// TIA Portal project "Funcoes" (V18)

(* hardware
DEVICE "S7-1200 station_1"  S7-1200 Station
   slot 0: "Rack_0"  S7-1200 Rack  Rack  V1.0
   slot 1: "PLC_1"  CPU 1214C AC/DC/Rly  6ES7 214-1BG40-0XB0  V4.5
   slot 2: "DI 16/DQ 16x24VDC_1"  6ES7 223-1BL32-0XB0  V2.0
   slot 3: "AI 8x13BIT_1"  6ES7 231-4HF32-0XB0  V2.1
*)

// ===== PLC "PLC_1"  CPU 1214C AC/DC/Rly =====

VAR_GLOBAL   // PLC tag table "Default tag table"
   "VC" AT %Q0.0 : Bool;
   "VT" AT %Q0.1 : Bool;
   "VD1" AT %Q0.2 : Bool;
   "VD2" AT %Q0.3 : Bool;
   "C1" AT %Q0.4 : Bool;
   "C2" AT %Q0.5 : Bool;
   "C3" AT %Q0.6 : Bool;
   "LED1" AT %Q0.7 : Bool;
   "LED2" AT %Q1.0 : Bool;
   "LE" AT %Q1.1 : Bool;
   "H" AT %Q8.0 : Bool;
   "BL" AT %I0.0 : Bool;
   "BD" AT %I0.1 : Bool;
   "BE" AT %I0.2 : Bool;
   "CS1" AT %I0.3 : Bool;
   "CS2" AT %I0.4 : Bool;
   "P" AT %IW112 : Int;
   "PS" AT %IW114 : Int;
   "PA" AT %IW116 : Int;
   "T" AT %IW118 : Int;
END_VAR

VAR_GLOBAL CONSTANT   // PLC tag table "Default tag table"
   "Lmin" : Real := 1.0;
   "L1" : Real := 1.5;
   "L2" : Real := 2.0;
   "Tlim" : Real := 0.6;
   "Ta" : Real := 2.0;
   "beta" : Real := 0.02;
   "Padm" : Real := 3.5;
   "Pmin" : Real := 0.1;
   "Peq" : Real := 3.0;
   "gamma" : Real := 0.01;
   "Plim" : Real := 0.1;
END_VAR

DATA_BLOCK "Data_block_1"   // DB1
{ S7_Optimized_Access := 'TRUE' }
VERSION : 0.1
   VAR
      n : Int := 0;
      "Valvulas ON" : Bool := false;
      "Valvulas ON - M3" : Bool := false;
      "Sequencia 1" : Array[0..2] of Int;
      "Sequencia 2" : Array[0..2] of Int;
      "Sequencia 3" : Array[0..2] of Int;
   END_VAR
   VAR RETAIN
      Sequencia : Array[0..2] of Int;
   END_VAR
   VAR
      "Tomada de decisao" : Bool := false;
      "Valores de pressao" : Array[0..9] of Real;
      index : Int := 0;
      "index max" : Int := 10;
      length : Int := 10;
      "Valores de pressao - M3" : Array[0..999] of Real;
      "index - M3" : Int := 0;
      "index max - M3" : Int := 1000;
      "length - M3" : Int := 0;
      "Atingir pressao eq" : Bool := false;
      "Plim atingida" : Bool := false;
      M2 : Bool := false;
      "Estado anterior" : Bool := false;
   END_VAR
BEGIN
   "Sequencia 1"[0] := 1;
   "Sequencia 1"[1] := 2;
   "Sequencia 1"[2] := 3;
   "Sequencia 2"[0] := 3;
   "Sequencia 2"[1] := 1;
   "Sequencia 2"[2] := 2;
   "Sequencia 3"[0] := 2;
   "Sequencia 3"[1] := 3;
   "Sequencia 3"[2] := 1;
   Sequencia[0] := 1;
   Sequencia[1] := 2;
   Sequencia[2] := 3;
   "Valores de pressao"[0] := 0.0;
   "Valores de pressao"[1] := 0.0;
   "Valores de pressao"[2] := 0.0;
   "Valores de pressao"[3] := 0.0;
   "Valores de pressao"[4] := 0.0;
   "Valores de pressao"[5] := 0.0;
   "Valores de pressao"[6] := 0.0;
   "Valores de pressao"[7] := 0.0;
   "Valores de pressao"[8] := 0.0;
   "Valores de pressao"[9] := 0.0;
END_DATA_BLOCK

// folder: System blocks/Program resources

DATA_BLOCK "Timer de amostragem"   // DB2
{ S7_Optimized_Access := 'TRUE' }
AUTHOR : Simatic
FAMILY : IEC
NAME : IEC_TMR
VERSION : 1.0
// stored: InstanceOfName IEC_TIMER
"IEC_TIMER"
BEGIN
   PT := T#1S;
END_DATA_BLOCK

DATA_BLOCK "Timer abastecimento"   // DB3
{ S7_Optimized_Access := 'TRUE' }
AUTHOR : Simatic
FAMILY : IEC
NAME : IEC_TMR
VERSION : 1.0
// stored: InstanceOfName IEC_TIMER
"IEC_TIMER"
BEGIN
   PT := T#1S;
END_DATA_BLOCK

// folder: (top level)

FUNCTION "Aciona valvulas - M1 e M2" : Void   // FC1, LAD
{ S7_Optimized_Access := 'TRUE' }
VERSION : 0.1
BEGIN

REGION Network 1: Acionando válvulas dos modos 1 e 2
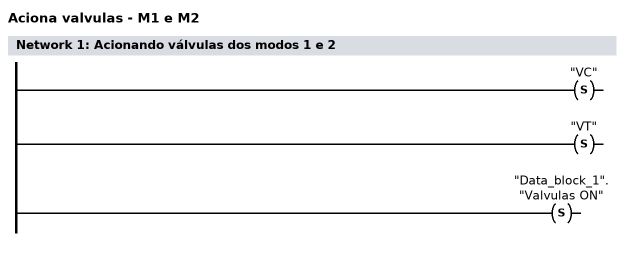
   RUNG wire#powerrail
      S_Coil( "VC" )
   END_RUNG
   RUNG wire#powerrail
      S_Coil( "VT" )
   END_RUNG
   RUNG wire#powerrail
      S_Coil( "Data_block_1"."Valvulas ON" )
   END_RUNG
   // the same network as SCL:
   "VC" := TRUE;
   "VT" := TRUE;
   "Data_block_1"."Valvulas ON" := TRUE;
END_REGION
END_FUNCTION

FUNCTION "Desliga valvulas - M1 e M2" : Void   // FC2, LAD
{ S7_Optimized_Access := 'TRUE' }
VERSION : 0.1
BEGIN

REGION Network 1: Válvula on/off da entrada do sistema de compressores
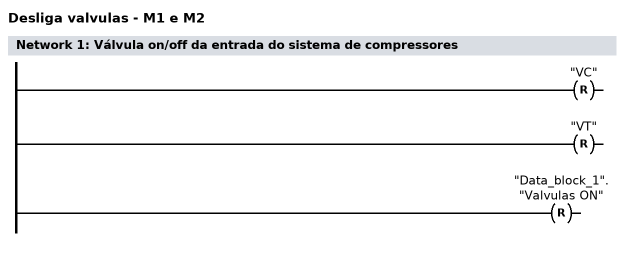
   RUNG wire#powerrail
      R_Coil( "VC" )
   END_RUNG
   RUNG wire#powerrail
      R_Coil( "VT" )
   END_RUNG
   RUNG wire#powerrail
      R_Coil( "Data_block_1"."Valvulas ON" )
   END_RUNG
   // the same network as SCL:
   "VC" := FALSE;
   "VT" := FALSE;
   "Data_block_1"."Valvulas ON" := FALSE;
END_REGION
END_FUNCTION

FUNCTION "Verifica valvulas 1" : Void   // FC3, LAD
{ S7_Optimized_Access := 'TRUE' }
VERSION : 0.1
BEGIN

REGION Network 1
   // Se válvulas OFF
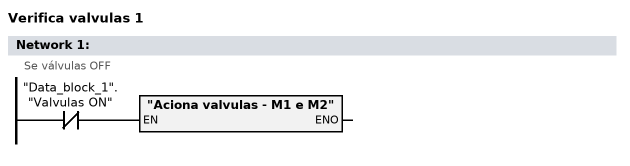
   RUNG wire#powerrail
      I_Contact( "Data_block_1"."Valvulas ON" )
      "Aciona valvulas - M1 e M2"()
   END_RUNG
   // the same network as SCL:
   IF NOT "Data_block_1"."Valvulas ON" THEN "Aciona valvulas - M1 e M2"(); END_IF;
END_REGION
END_FUNCTION

FUNCTION "Verifica valvulas 2" : Void   // FC4, LAD
{ S7_Optimized_Access := 'TRUE' }
VERSION : 0.1
BEGIN

REGION Network 1
   // Se válvulas ON
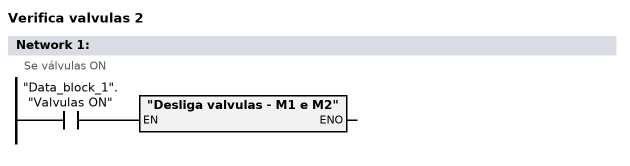
   RUNG wire#powerrail
      Contact( "Data_block_1"."Valvulas ON" )
      "Desliga valvulas - M1 e M2"()
   END_RUNG
   // the same network as SCL:
   IF "Data_block_1"."Valvulas ON" THEN "Desliga valvulas - M1 e M2"(); END_IF;
END_REGION
END_FUNCTION

FUNCTION "Obtem pressao" : Void   // FC5, LAD
{ S7_Optimized_Access := 'TRUE' }
VERSION : 0.1
   VAR_OUTPUT
      Pressao : Real;   // Pressão obtida
   END_VAR
   VAR_TEMP
      "Pressao normalizada" : Real;   // Pressão normalizada
   END_VAR
BEGIN

REGION Network 1
   // Normalização do valor de pressão lido do transmissor
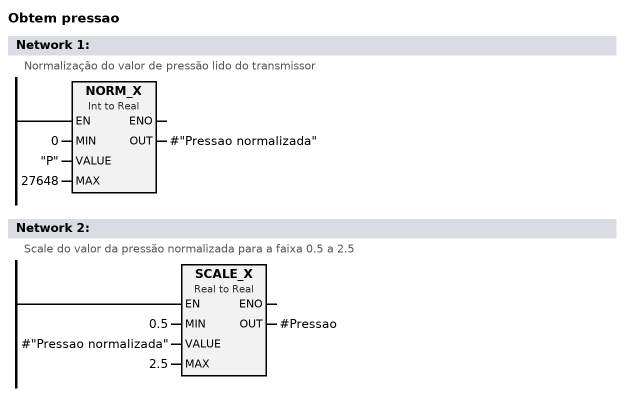
   RUNG wire#powerrail
      { S7_Templates := "[SrcType := Int, DestType := Real]" } Normalize(min := 0, value := "P", max := 27648, out => #"Pressao normalizada")
   END_RUNG
   // the same network as SCL:
   #"Pressao normalizada" := NORM_X(MIN := 0, VALUE := "P", MAX := 27648);
END_REGION

REGION Network 2
   // Scale do valor da pressão normalizada para a faixa 0.5 a 2.5
   RUNG wire#powerrail
      { S7_Templates := "[SrcType := Real, DestType := Real]" } Scale(min := 0.5, value := #"Pressao normalizada", max := 2.5, out => #Pressao)
   END_RUNG
   // the same network as SCL:
   #Pressao := SCALE_X(MIN := 0.5, VALUE := #"Pressao normalizada", MAX := 2.5);
END_REGION
END_FUNCTION

FUNCTION "Pressao crescente" : Void   // FC6, LAD
{ S7_Optimized_Access := 'TRUE' }
VERSION : 0.1
   VAR_INPUT
      P : Real;   // Pressão no interior do tanque separador
   END_VAR
   VAR_TEMP   // added for the SCL form of the ladder/FBD networks
      _w1 : Bool;
      _w2 : Bool;
   END_VAR
BEGIN

REGION Network 1
   // Se pressão entre Lmin e L1
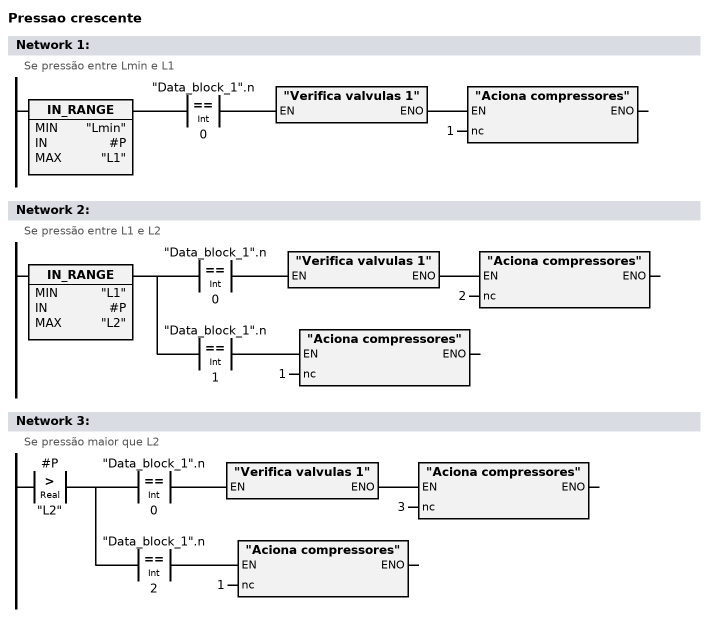
   RUNG wire#powerrail
      { S7_Templates := "SrcType := Real" } InRange(min := "Lmin", in := #P, max := "L1")
      { S7_Templates := "SrcType := Int" } EQ_Contact(in1 := "Data_block_1".n, in2 := 0)
      "Verifica valvulas 1"()
      "Aciona compressores"(nc := 1)
   END_RUNG
   // the same network as SCL:
   "Verifica valvulas 1"(EN := ("Lmin" <= #P) AND (#P <= "L1") AND ("Data_block_1".n = 0), ENO => #_w1);
   IF #_w1 THEN "Aciona compressores"(nc := 1); END_IF;
END_REGION

REGION Network 2
   // Se pressão entre L1 e L2
   RUNG wire#powerrail
      { S7_Templates := "SrcType := Real" } InRange(min := "L1", in := #P, max := "L2")
      wire#w1
      { S7_Templates := "SrcType := Int" } EQ_Contact(in1 := "Data_block_1".n, in2 := 0)
      "Verifica valvulas 1"()
      "Aciona compressores"(nc := 2)
   END_RUNG
   RUNG wire#w1
      { S7_Templates := "SrcType := Int" } EQ_Contact(in1 := "Data_block_1".n, in2 := 1)
      "Aciona compressores"(nc := 1)
   END_RUNG
   // the same network as SCL:
   #_w1 := ("L1" <= #P) AND (#P <= "L2");
   "Verifica valvulas 1"(EN := #_w1 AND ("Data_block_1".n = 0), ENO => #_w2);
   IF #_w2 THEN "Aciona compressores"(nc := 2); END_IF;
   IF #_w1 AND ("Data_block_1".n = 1) THEN "Aciona compressores"(nc := 1); END_IF;
END_REGION

REGION Network 3
   // Se pressão maior que L2
   RUNG wire#powerrail
      { S7_Templates := "SrcType := Real" } GT_Contact(in1 := #P, in2 := "L2")
      wire#w1
      { S7_Templates := "SrcType := Int" } EQ_Contact(in1 := "Data_block_1".n, in2 := 0)
      "Verifica valvulas 1"()
      "Aciona compressores"(nc := 3)
   END_RUNG
   RUNG wire#w1
      { S7_Templates := "SrcType := Int" } EQ_Contact(in1 := "Data_block_1".n, in2 := 2)
      "Aciona compressores"(nc := 1)
   END_RUNG
   // the same network as SCL:
   #_w1 := #P > "L2";
   "Verifica valvulas 1"(EN := #_w1 AND ("Data_block_1".n = 0), ENO => #_w2);
   IF #_w2 THEN "Aciona compressores"(nc := 3); END_IF;
   IF #_w1 AND ("Data_block_1".n = 2) THEN "Aciona compressores"(nc := 1); END_IF;
END_REGION
END_FUNCTION

FUNCTION "Pressao decrescente" : Void   // FC7, LAD
{ S7_Optimized_Access := 'TRUE' }
VERSION : 0.1
   VAR_INPUT
      P : Real;   // Pressão no interior do tanque separador
   END_VAR
   VAR_TEMP   // added for the SCL form of the ladder/FBD networks
      _w1 : Bool;
   END_VAR
BEGIN

REGION Network 1
   // Se pressão entre L1 e L2
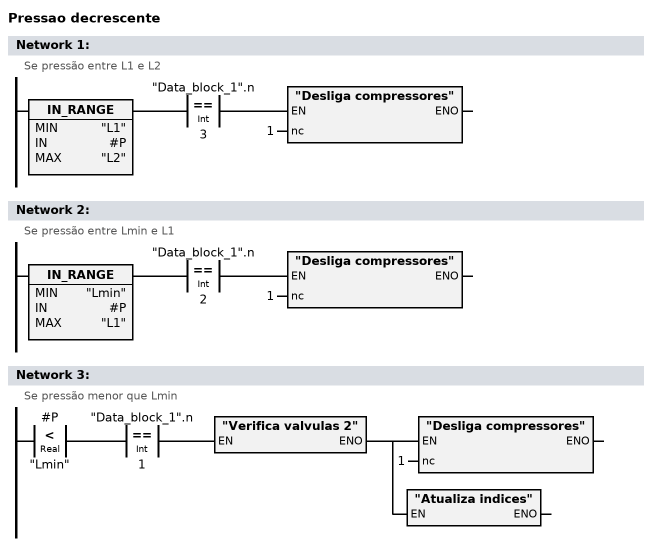
   RUNG wire#powerrail
      { S7_Templates := "SrcType := Real" } InRange(min := "L1", in := #P, max := "L2")
      { S7_Templates := "SrcType := Int" } EQ_Contact(in1 := "Data_block_1".n, in2 := 3)
      "Desliga compressores"(nc := 1)
   END_RUNG
   // the same network as SCL:
   IF ("L1" <= #P) AND (#P <= "L2") AND ("Data_block_1".n = 3) THEN "Desliga compressores"(nc := 1); END_IF;
END_REGION

REGION Network 2
   // Se pressão entre Lmin e L1
   RUNG wire#powerrail
      { S7_Templates := "SrcType := Real" } InRange(min := "Lmin", in := #P, max := "L1")
      { S7_Templates := "SrcType := Int" } EQ_Contact(in1 := "Data_block_1".n, in2 := 2)
      "Desliga compressores"(nc := 1)
   END_RUNG
   // the same network as SCL:
   IF ("Lmin" <= #P) AND (#P <= "L1") AND ("Data_block_1".n = 2) THEN
       "Desliga compressores"(nc := 1);
   END_IF;
END_REGION

REGION Network 3
   // Se pressão menor que Lmin
   RUNG wire#powerrail
      { S7_Templates := "SrcType := Real" } LT_Contact(in1 := #P, in2 := "Lmin")
      { S7_Templates := "SrcType := Int" } EQ_Contact(in1 := "Data_block_1".n, in2 := 1)
      "Verifica valvulas 2"()
      wire#w1
      "Desliga compressores"(nc := 1)
   END_RUNG
   RUNG wire#w1
      "Atualiza indices"()
   END_RUNG
   // the same network as SCL:
   "Verifica valvulas 2"(EN := (#P < "Lmin") AND ("Data_block_1".n = 1), ENO => #_w1);
   IF #_w1 THEN
       "Desliga compressores"(nc := 1);
       "Atualiza indices"();
   END_IF;
END_REGION
END_FUNCTION

FUNCTION "Aciona compressores" : Void   // FC8, LAD
{ S7_Optimized_Access := 'TRUE' }
VERSION : 0.1
   VAR_INPUT
      nc : Int;   // Número de compressores
   END_VAR
   VAR_TEMP   // added for the SCL form of the ladder/FBD networks
      _w1 : Bool;
      _w2 : Bool;
      _w3 : Bool;
      _w4 : Bool;
   END_VAR
BEGIN

REGION Network 1
   // Apenas um compressor deve ser ligado
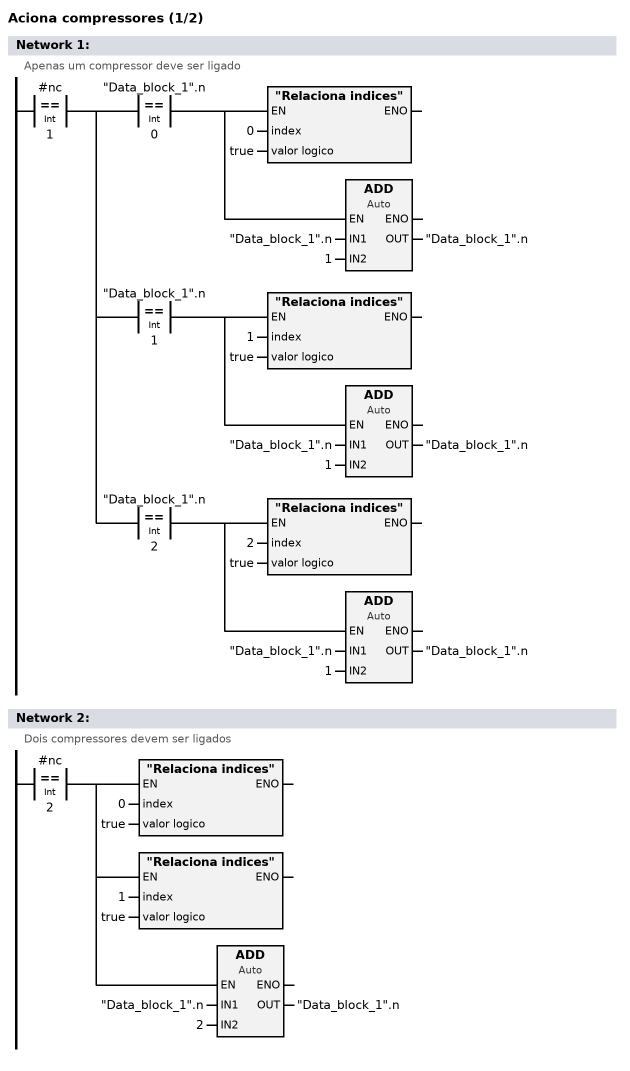
   RUNG wire#powerrail
      { S7_Templates := "SrcType := Int" } EQ_Contact(in1 := #nc, in2 := 1)
      wire#w1
      { S7_Templates := "SrcType := Int" } EQ_Contact(in1 := "Data_block_1".n, in2 := 0)
      wire#w2
      "Relaciona indices"(index := 0, "valor logico" := true)
   END_RUNG
   RUNG wire#w2
      Add(in1 := "Data_block_1".n, in2 := 1, out => "Data_block_1".n)
   END_RUNG
   RUNG wire#w1
      { S7_Templates := "SrcType := Int" } EQ_Contact(in1 := "Data_block_1".n, in2 := 1)
      wire#w3
      "Relaciona indices"(index := 1, "valor logico" := true)
   END_RUNG
   RUNG wire#w3
      Add(in1 := "Data_block_1".n, in2 := 1, out => "Data_block_1".n)
   END_RUNG
   RUNG wire#w1
      { S7_Templates := "SrcType := Int" } EQ_Contact(in1 := "Data_block_1".n, in2 := 2)
      wire#w4
      "Relaciona indices"(index := 2, "valor logico" := true)
   END_RUNG
   RUNG wire#w4
      Add(in1 := "Data_block_1".n, in2 := 1, out => "Data_block_1".n)
   END_RUNG
   // the same network as SCL:
   #_w1 := #nc = 1;
   #_w2 := #_w1 AND ("Data_block_1".n = 0);
   IF #_w2 THEN
       "Relaciona indices"(index := 0, "valor logico" := true);
       "Data_block_1".n := "Data_block_1".n + 1;
   END_IF;
   #_w3 := #_w1 AND ("Data_block_1".n = 1);
   IF #_w3 THEN
       "Relaciona indices"(index := 1, "valor logico" := true);
       "Data_block_1".n := "Data_block_1".n + 1;
   END_IF;
   #_w4 := #_w1 AND ("Data_block_1".n = 2);
   IF #_w4 THEN
       "Relaciona indices"(index := 2, "valor logico" := true);
       "Data_block_1".n := "Data_block_1".n + 1;
   END_IF;
END_REGION

REGION Network 2
   // Dois compressores devem ser ligados
   RUNG wire#powerrail
      { S7_Templates := "SrcType := Int" } EQ_Contact(in1 := #nc, in2 := 2)
      wire#w1
      "Relaciona indices"(index := 0, "valor logico" := true)
   END_RUNG
   RUNG wire#w1
      "Relaciona indices"(index := 1, "valor logico" := true)
   END_RUNG
   RUNG wire#w1
      Add(in1 := "Data_block_1".n, in2 := 2, out => "Data_block_1".n)
   END_RUNG
   // the same network as SCL:
   IF #nc = 2 THEN
       "Relaciona indices"(index := 0, "valor logico" := true);
       "Relaciona indices"(index := 1, "valor logico" := true);
       "Data_block_1".n := "Data_block_1".n + 2;
   END_IF;
END_REGION

REGION Network 3
   // Três compressores devem ser ligados
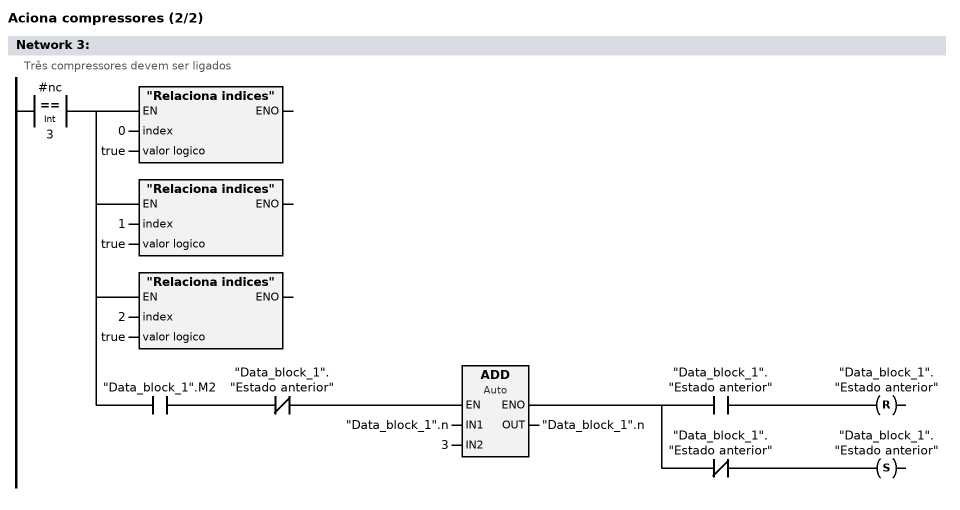
   RUNG wire#powerrail
      { S7_Templates := "SrcType := Int" } EQ_Contact(in1 := #nc, in2 := 3)
      wire#w1
      "Relaciona indices"(index := 0, "valor logico" := true)
   END_RUNG
   RUNG wire#w1
      "Relaciona indices"(index := 1, "valor logico" := true)
   END_RUNG
   RUNG wire#w1
      "Relaciona indices"(index := 2, "valor logico" := true)
   END_RUNG
   RUNG wire#w1
      Contact( "Data_block_1".M2 )
      I_Contact( "Data_block_1"."Estado anterior" )
      Add(in1 := "Data_block_1".n, in2 := 3, out => "Data_block_1".n)
      wire#w2
      Contact( "Data_block_1"."Estado anterior" )
      R_Coil( "Data_block_1"."Estado anterior" )
   END_RUNG
   RUNG wire#w2
      I_Contact( "Data_block_1"."Estado anterior" )
      S_Coil( "Data_block_1"."Estado anterior" )
   END_RUNG
   // the same network as SCL:
   #_w1 := #nc = 3;
   IF #_w1 THEN
       "Relaciona indices"(index := 0, "valor logico" := true);
       "Relaciona indices"(index := 1, "valor logico" := true);
       "Relaciona indices"(index := 2, "valor logico" := true);
   END_IF;
   #_w2 := #_w1 AND "Data_block_1".M2 AND NOT "Data_block_1"."Estado anterior";
   IF #_w2 THEN "Data_block_1".n := "Data_block_1".n + 3; END_IF;
   IF #_w2 AND "Data_block_1"."Estado anterior" THEN "Data_block_1"."Estado anterior" := FALSE; END_IF;
   IF #_w2 AND NOT "Data_block_1"."Estado anterior" THEN "Data_block_1"."Estado anterior" := TRUE; END_IF;
END_REGION
END_FUNCTION

FUNCTION "Desliga compressores" : Void   // FC9, LAD
{ S7_Optimized_Access := 'TRUE' }
VERSION : 0.1
   VAR_INPUT
      nc : Int;   // Número de compressores
   END_VAR
   VAR_TEMP   // added for the SCL form of the ladder/FBD networks
      _w1 : Bool;
      _w2 : Bool;
      _w3 : Bool;
      _w4 : Bool;
   END_VAR
BEGIN

REGION Network 1
   // Apenas um compressor deve ser desligado
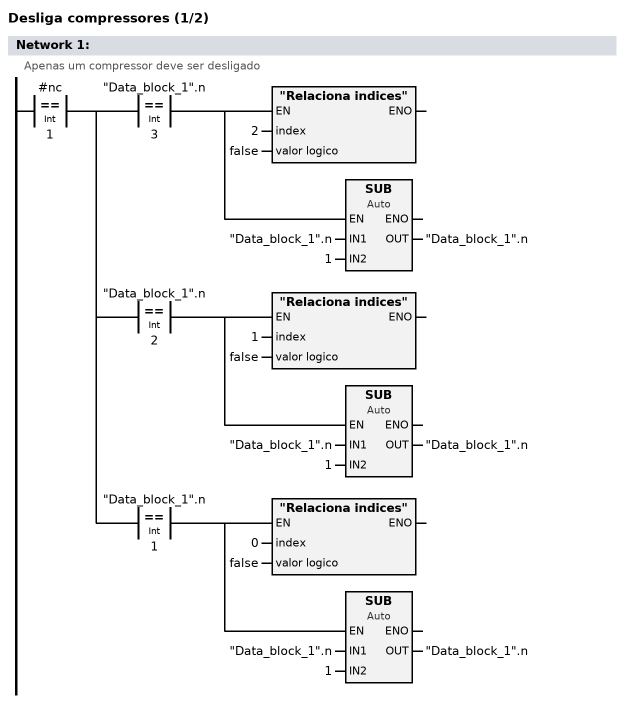
   RUNG wire#powerrail
      { S7_Templates := "SrcType := Int" } EQ_Contact(in1 := #nc, in2 := 1)
      wire#w1
      { S7_Templates := "SrcType := Int" } EQ_Contact(in1 := "Data_block_1".n, in2 := 3)
      wire#w2
      "Relaciona indices"(index := 2, "valor logico" := false)
   END_RUNG
   RUNG wire#w2
      Sub(in1 := "Data_block_1".n, in2 := 1, out => "Data_block_1".n)
   END_RUNG
   RUNG wire#w1
      { S7_Templates := "SrcType := Int" } EQ_Contact(in1 := "Data_block_1".n, in2 := 2)
      wire#w3
      "Relaciona indices"(index := 1, "valor logico" := false)
   END_RUNG
   RUNG wire#w3
      Sub(in1 := "Data_block_1".n, in2 := 1, out => "Data_block_1".n)
   END_RUNG
   RUNG wire#w1
      { S7_Templates := "SrcType := Int" } EQ_Contact(in1 := "Data_block_1".n, in2 := 1)
      wire#w4
      "Relaciona indices"(index := 0, "valor logico" := false)
   END_RUNG
   RUNG wire#w4
      Sub(in1 := "Data_block_1".n, in2 := 1, out => "Data_block_1".n)
   END_RUNG
   // the same network as SCL:
   #_w1 := #nc = 1;
   #_w2 := #_w1 AND ("Data_block_1".n = 3);
   IF #_w2 THEN
       "Relaciona indices"(index := 2, "valor logico" := false);
       "Data_block_1".n := "Data_block_1".n - 1;
   END_IF;
   #_w3 := #_w1 AND ("Data_block_1".n = 2);
   IF #_w3 THEN
       "Relaciona indices"(index := 1, "valor logico" := false);
       "Data_block_1".n := "Data_block_1".n - 1;
   END_IF;
   #_w4 := #_w1 AND ("Data_block_1".n = 1);
   IF #_w4 THEN
       "Relaciona indices"(index := 0, "valor logico" := false);
       "Data_block_1".n := "Data_block_1".n - 1;
   END_IF;
END_REGION

REGION Network 2
   // Devem ser desligados todos os compressores que estiverem ligados
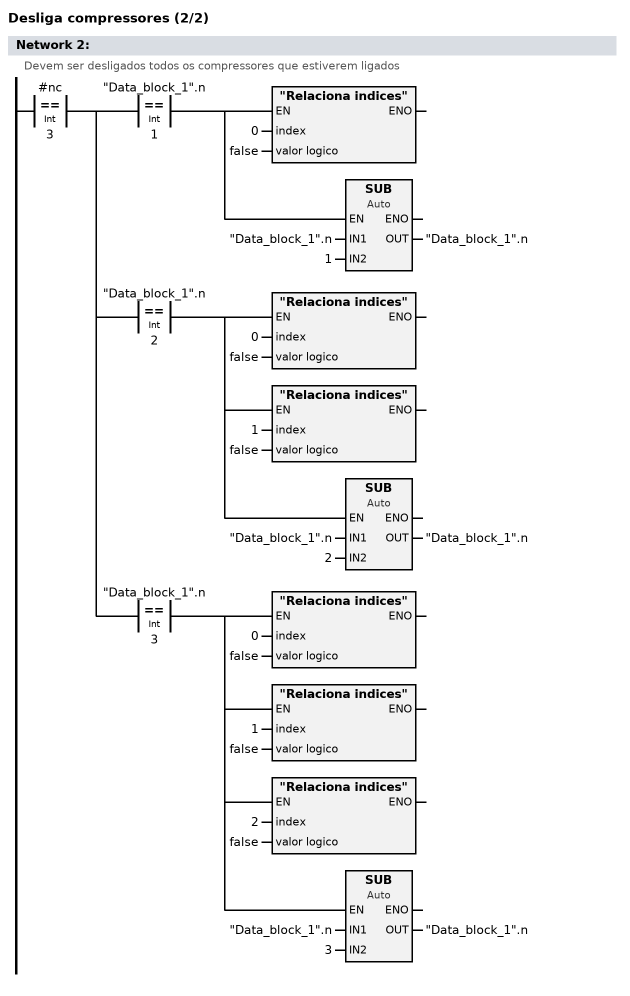
   RUNG wire#powerrail
      { S7_Templates := "SrcType := Int" } EQ_Contact(in1 := #nc, in2 := 3)
      wire#w1
      { S7_Templates := "SrcType := Int" } EQ_Contact(in1 := "Data_block_1".n, in2 := 1)
      wire#w2
      "Relaciona indices"(index := 0, "valor logico" := false)
   END_RUNG
   RUNG wire#w2
      Sub(in1 := "Data_block_1".n, in2 := 1, out => "Data_block_1".n)
   END_RUNG
   RUNG wire#w1
      { S7_Templates := "SrcType := Int" } EQ_Contact(in1 := "Data_block_1".n, in2 := 2)
      wire#w3
      "Relaciona indices"(index := 0, "valor logico" := false)
   END_RUNG
   RUNG wire#w3
      "Relaciona indices"(index := 1, "valor logico" := false)
   END_RUNG
   RUNG wire#w3
      Sub(in1 := "Data_block_1".n, in2 := 2, out => "Data_block_1".n)
   END_RUNG
   RUNG wire#w1
      { S7_Templates := "SrcType := Int" } EQ_Contact(in1 := "Data_block_1".n, in2 := 3)
      wire#w4
      "Relaciona indices"(index := 0, "valor logico" := false)
   END_RUNG
   RUNG wire#w4
      "Relaciona indices"(index := 1, "valor logico" := false)
   END_RUNG
   RUNG wire#w4
      "Relaciona indices"(index := 2, "valor logico" := false)
   END_RUNG
   RUNG wire#w4
      Sub(in1 := "Data_block_1".n, in2 := 3, out => "Data_block_1".n)
   END_RUNG
   // the same network as SCL:
   #_w1 := #nc = 3;
   #_w2 := #_w1 AND ("Data_block_1".n = 1);
   IF #_w2 THEN
       "Relaciona indices"(index := 0, "valor logico" := false);
       "Data_block_1".n := "Data_block_1".n - 1;
   END_IF;
   #_w3 := #_w1 AND ("Data_block_1".n = 2);
   IF #_w3 THEN
       "Relaciona indices"(index := 0, "valor logico" := false);
       "Relaciona indices"(index := 1, "valor logico" := false);
       "Data_block_1".n := "Data_block_1".n - 2;
   END_IF;
   #_w4 := #_w1 AND ("Data_block_1".n = 3);
   IF #_w4 THEN
       "Relaciona indices"(index := 0, "valor logico" := false);
       "Relaciona indices"(index := 1, "valor logico" := false);
       "Relaciona indices"(index := 2, "valor logico" := false);
       "Data_block_1".n := "Data_block_1".n - 3;
   END_IF;
END_REGION
END_FUNCTION

FUNCTION "Verifica compressores" : Void   // FC10, LAD
{ S7_Optimized_Access := 'TRUE' }
VERSION : 0.1
BEGIN

REGION Network 1
   // Se houver algum compressor acionado
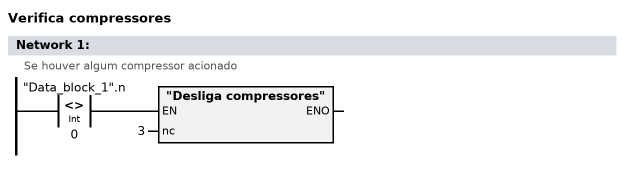
   RUNG wire#powerrail
      { S7_Templates := "SrcType := Int" } NE_Contact(in1 := "Data_block_1".n, in2 := 0)
      "Desliga compressores"(nc := 3)
   END_RUNG
   // the same network as SCL:
   IF "Data_block_1".n <> 0 THEN "Desliga compressores"(nc := 3); END_IF;
END_REGION
END_FUNCTION

FUNCTION "Finaliza operacao" : Void   // FC11, LAD
{ S7_Optimized_Access := 'TRUE' }
VERSION : 0.1
BEGIN

REGION Network 1
   // Finalizando operação
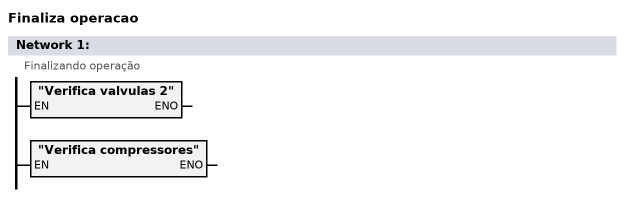
   RUNG wire#powerrail
      "Verifica valvulas 2"()
   END_RUNG
   RUNG wire#powerrail
      "Verifica compressores"()
   END_RUNG
   // the same network as SCL:
   "Verifica valvulas 2"();
   "Verifica compressores"();
END_REGION
END_FUNCTION

FUNCTION "M2 - Operacao iniciada" : Void   // FC12, LAD
{ S7_Optimized_Access := 'TRUE' }
VERSION : 0.1
   VAR_TEMP   // added for the SCL form of the ladder/FBD networks
      _w1 : Bool;
   END_VAR
BEGIN

REGION Network 1
   // MODO MANUAL [M2] - Operação iniciada
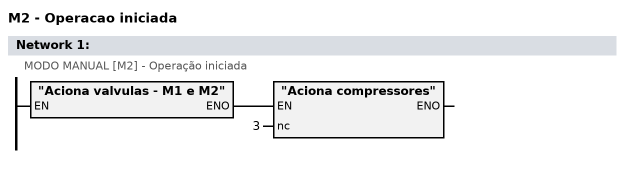
   RUNG wire#powerrail
      "Aciona valvulas - M1 e M2"()
      "Aciona compressores"(nc := 3)
   END_RUNG
   // the same network as SCL:
   "Aciona valvulas - M1 e M2"(ENO => #_w1);
   IF #_w1 THEN "Aciona compressores"(nc := 3); END_IF;
END_REGION
END_FUNCTION

FUNCTION "M2 - Operacao finalizada" : Void   // FC13, LAD
{ S7_Optimized_Access := 'TRUE' }
VERSION : 0.1
BEGIN

REGION Network 1
   // MODO MANUAL [M2] - Operação finalizada
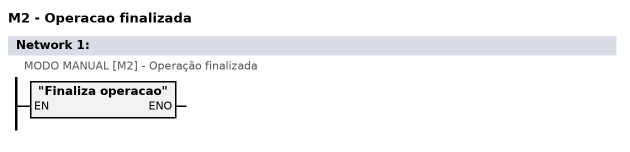
   RUNG wire#powerrail
      "Finaliza operacao"()
   END_RUNG
   // the same network as SCL:
   "Finaliza operacao"();
END_REGION
END_FUNCTION

FUNCTION "Aciona valvulas - M3" : Void   // FC14, LAD
{ S7_Optimized_Access := 'TRUE' }
VERSION : 0.1
BEGIN

REGION Network 1
   // Acionando válvulas da linha direta
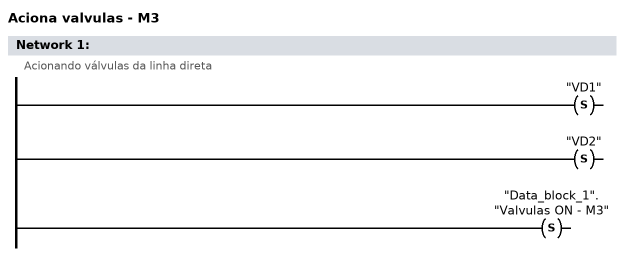
   RUNG wire#powerrail
      S_Coil( "VD1" )
   END_RUNG
   RUNG wire#powerrail
      S_Coil( "VD2" )
   END_RUNG
   RUNG wire#powerrail
      S_Coil( "Data_block_1"."Valvulas ON - M3" )
   END_RUNG
   // the same network as SCL:
   "VD1" := TRUE;
   "VD2" := TRUE;
   "Data_block_1"."Valvulas ON - M3" := TRUE;
END_REGION
END_FUNCTION

FUNCTION "Obtem temperatura" : Void   // FC15, LAD
{ S7_Optimized_Access := 'TRUE' }
VERSION : 0.1
   VAR_OUTPUT
      Temperatura : Real;   // Temperatura obtida
   END_VAR
   VAR_TEMP
      "Temperatura normalizada" : Real;   // Temperatura normalizada
   END_VAR
BEGIN

REGION Network 1
   // Normalização do valor de temperatura lido do transmissor
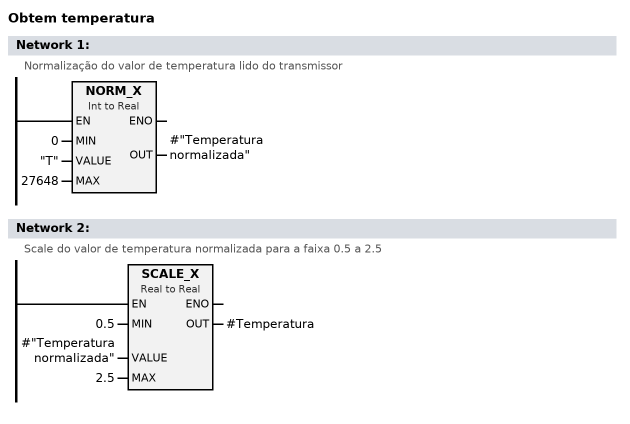
   RUNG wire#powerrail
      { S7_Templates := "[SrcType := Int, DestType := Real]" } Normalize(min := 0, value := "T", max := 27648, out => #"Temperatura normalizada")
   END_RUNG
   // the same network as SCL:
   #"Temperatura normalizada" := NORM_X(MIN := 0, VALUE := "T", MAX := 27648);
END_REGION

REGION Network 2
   // Scale do valor de temperatura normalizada para a faixa 0.5 a 2.5
   RUNG wire#powerrail
      { S7_Templates := "[SrcType := Real, DestType := Real]" } Scale(min := 0.5, value := #"Temperatura normalizada", max := 2.5, out => #Temperatura)
   END_RUNG
   // the same network as SCL:
   #Temperatura := SCALE_X(MIN := 0.5, VALUE := #"Temperatura normalizada", MAX := 2.5);
END_REGION
END_FUNCTION

FUNCTION "Atinge pressao de eq" : Void   // FC16, LAD
{ S7_Optimized_Access := 'TRUE' }
VERSION : 0.1
   VAR_TEMP
      "Threshold de Ta" : Real;   // Threshold da temperatura ambiente
      Temperatura : Real;   // Temperatura obtida
   END_VAR
   VAR_TEMP   // added for the SCL form of the ladder/FBD networks
      _w1 : Bool;
   END_VAR
BEGIN

REGION Network 1
   // Monitora temperatura
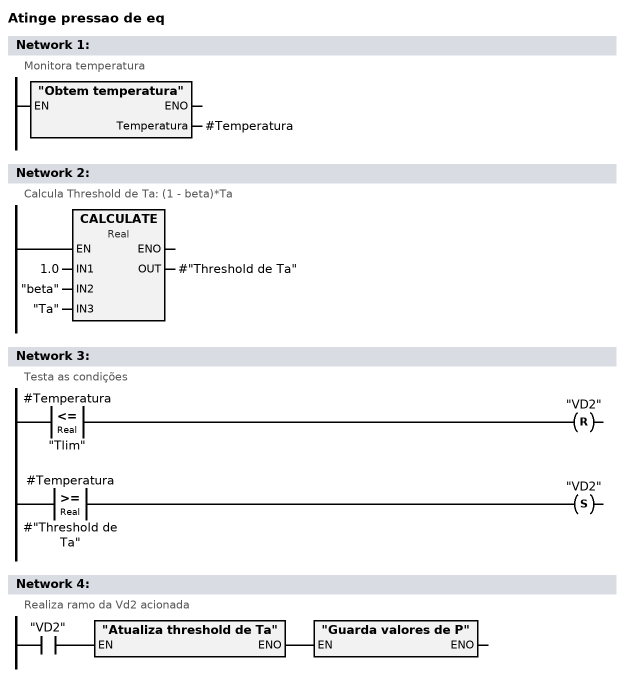
   RUNG wire#powerrail
      "Obtem temperatura"(Temperatura => #Temperatura)
   END_RUNG
   // the same network as SCL:
   "Obtem temperatura"(Temperatura => #Temperatura);
END_REGION

REGION Network 2
   // Calcula Threshold de Ta: (1 - beta)*Ta
   RUNG wire#powerrail
      { S7_Templates := "SrcType := Real"; S7_Expression := "(IN1 - IN2) * IN3" } Calculate(in1 := 1.0, in2 := "beta", in3 := "Ta", out => #"Threshold de Ta")
   END_RUNG
   // the same network as SCL:
   #"Threshold de Ta" := (1.0 - "beta") * "Ta";
END_REGION

REGION Network 3
   // Testa as condições
   RUNG wire#powerrail
      { S7_Templates := "SrcType := Real" } LE_Contact(in1 := #Temperatura, in2 := "Tlim")
      R_Coil( "VD2" )
   END_RUNG
   RUNG wire#powerrail
      { S7_Templates := "SrcType := Real" } GE_Contact(in1 := #Temperatura, in2 := #"Threshold de Ta")
      S_Coil( "VD2" )
   END_RUNG
   // the same network as SCL:
   IF #Temperatura <= "Tlim" THEN "VD2" := FALSE; END_IF;
   IF #Temperatura >= #"Threshold de Ta" THEN "VD2" := TRUE; END_IF;
END_REGION

REGION Network 4
   // Realiza ramo da Vd2 acionada
   RUNG wire#powerrail
      Contact( "VD2" )
      "Atualiza threshold de Ta"()
      "Guarda valores de P"()
   END_RUNG
   // the same network as SCL:
   "Atualiza threshold de Ta"(EN := "VD2", ENO => #_w1);
   IF #_w1 THEN "Guarda valores de P"(); END_IF;
END_REGION
END_FUNCTION

FUNCTION "Atualiza threshold de Ta" : Void   // FC17, LAD
{ S7_Optimized_Access := 'TRUE' }
VERSION : 0.1
BEGIN
END_FUNCTION

FUNCTION "Guarda valores de P" : Void   // FC18, LAD
{ S7_Optimized_Access := 'TRUE' }
VERSION : 0.1
   VAR_TEMP
      "Pressao abastecimento" : Real;
   END_VAR
BEGIN

REGION Network 1
   // Obtém pressão do nó estendido
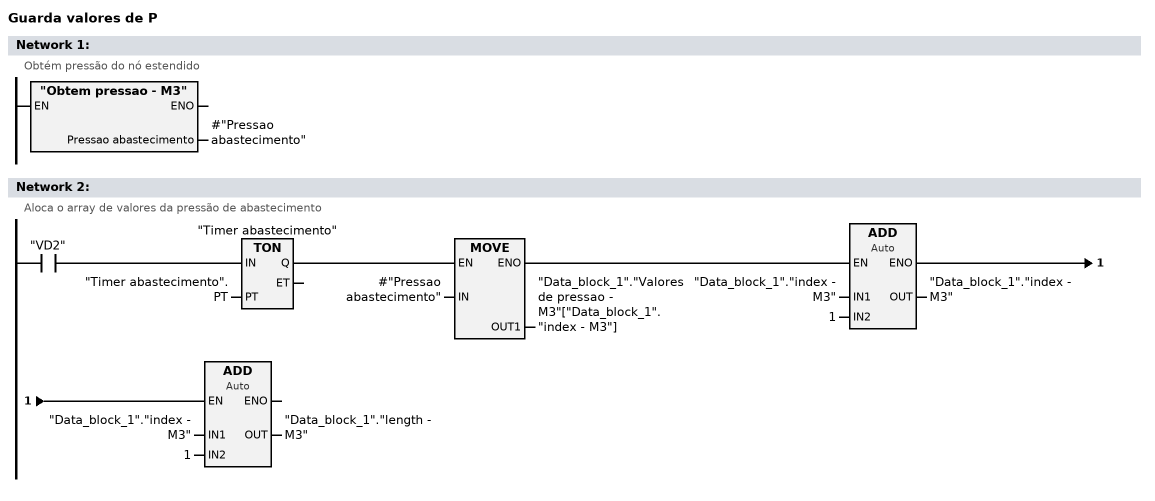
   RUNG wire#powerrail
      "Obtem pressao - M3"("Pressao abastecimento" => #"Pressao abastecimento")
   END_RUNG
   // the same network as SCL:
   "Obtem pressao - M3"("Pressao abastecimento" => #"Pressao abastecimento");
END_REGION

REGION Network 2
   // Aloca o array de valores da pressão de abastecimento
   "Timer abastecimento".TON(IN := "VD2", PT := "Timer abastecimento".PT);
   IF "Timer abastecimento".Q THEN
       "Data_block_1"."Valores de pressao - M3"["Data_block_1"."index - M3"] := #"Pressao abastecimento";
       "Data_block_1"."index - M3" := "Data_block_1"."index - M3" + 1;
       "Data_block_1"."length - M3" := "Data_block_1"."index - M3" + 1;
   END_IF;
END_REGION
END_FUNCTION

FUNCTION "Protocolo de Emergencia" : Void   // FC19, LAD
{ S7_Optimized_Access := 'TRUE' }
VERSION : 0.1
BEGIN

REGION Network 1
   // Aciona LED de emergência e alarme H
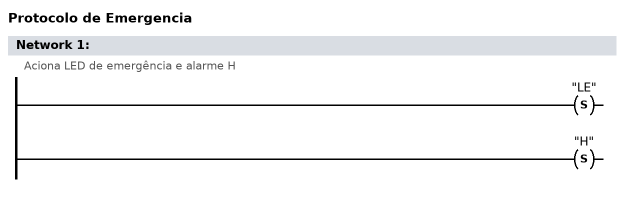
   RUNG wire#powerrail
      S_Coil( "LE" )
   END_RUNG
   RUNG wire#powerrail
      S_Coil( "H" )
   END_RUNG
   // the same network as SCL:
   "LE" := TRUE;
   "H" := TRUE;
END_REGION
END_FUNCTION

FUNCTION "OPERACAO - M2" : Void   // FC20, LAD
{ S7_Optimized_Access := 'TRUE' }
VERSION : 0.1
   VAR_TEMP   // added for the SCL form of the ladder/FBD networks
      _w1 : Bool;
   END_VAR
BEGIN

REGION Network 1
   // Em operação
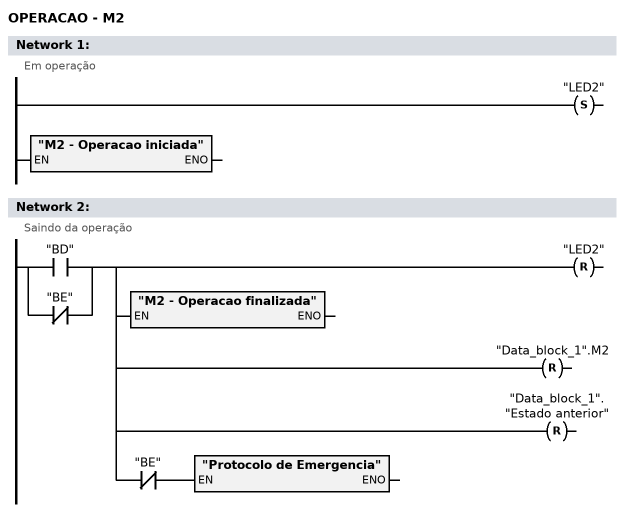
   RUNG wire#powerrail
      S_Coil( "LED2" )
   END_RUNG
   RUNG wire#powerrail
      "M2 - Operacao iniciada"()
   END_RUNG
   // the same network as SCL:
   "LED2" := TRUE;
   "M2 - Operacao iniciada"();
END_REGION

REGION Network 2
   // Saindo da operação
   RUNG wire#powerrail
      Contact( "BD" )
      wire#w1
      R_Coil( "LED2" )
   END_RUNG
   RUNG wire#powerrail
      I_Contact( "BE" )
   END_RUNG wire#w1
   RUNG wire#w1
      "M2 - Operacao finalizada"()
   END_RUNG
   RUNG wire#w1
      R_Coil( "Data_block_1".M2 )
   END_RUNG
   RUNG wire#w1
      R_Coil( "Data_block_1"."Estado anterior" )
   END_RUNG
   RUNG wire#w1
      I_Contact( "BE" )
      "Protocolo de Emergencia"()
   END_RUNG
   // the same network as SCL:
   #_w1 := "BD" OR NOT "BE";
   IF #_w1 THEN
       "LED2" := FALSE;
       "M2 - Operacao finalizada"();
       "Data_block_1".M2 := FALSE;
       "Data_block_1"."Estado anterior" := FALSE;
   END_IF;
   IF #_w1 AND NOT "BE" THEN "Protocolo de Emergencia"(); END_IF;
END_REGION
END_FUNCTION

FUNCTION "Logica CONJUNTA" : Void   // FC21, LAD
{ S7_Optimized_Access := 'TRUE' }
VERSION : 0.1
   VAR_TEMP
      Pressao : Real;   // Pressão obtida
   END_VAR
BEGIN

REGION Network 1
   // Chave seletora na posição 1
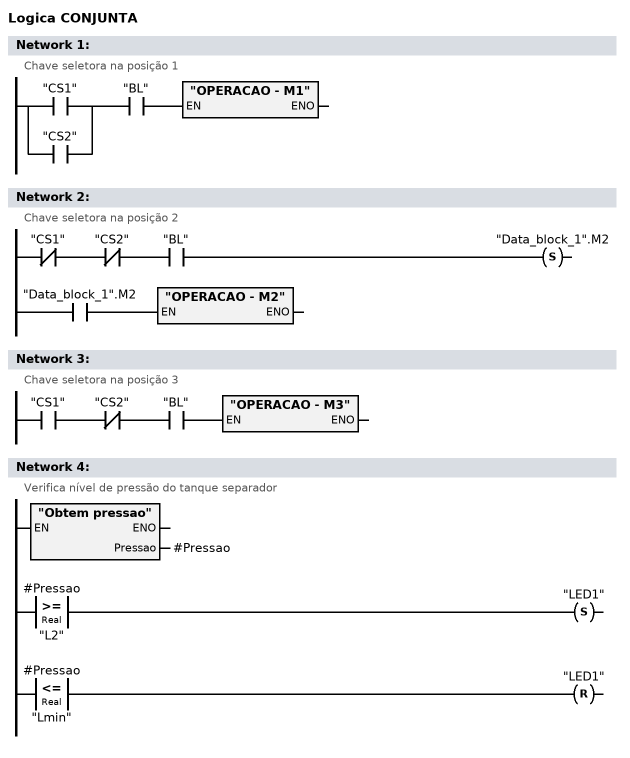
   RUNG wire#powerrail
      Contact( "CS1" )
      wire#w1
      Contact( "BL" )
      "OPERACAO - M1"()
   END_RUNG
   RUNG wire#powerrail
      Contact( "CS2" )
   END_RUNG wire#w1
   // the same network as SCL:
   IF ("CS1" OR "CS2") AND "BL" THEN "OPERACAO - M1"(); END_IF;
END_REGION

REGION Network 2
   // Chave seletora na posição 2
   RUNG wire#powerrail
      I_Contact( "CS1" )
      I_Contact( "CS2" )
      Contact( "BL" )
      S_Coil( "Data_block_1".M2 )
   END_RUNG
   RUNG wire#powerrail
      Contact( "Data_block_1".M2 )
      "OPERACAO - M2"()
   END_RUNG
   // the same network as SCL:
   IF NOT "CS1" AND NOT "CS2" AND "BL" THEN "Data_block_1".M2 := TRUE; END_IF;
   IF "Data_block_1".M2 THEN "OPERACAO - M2"(); END_IF;
END_REGION

REGION Network 3
   // Chave seletora na posição 3
   RUNG wire#powerrail
      Contact( "CS1" )
      I_Contact( "CS2" )
      Contact( "BL" )
      "OPERACAO - M3"()
   END_RUNG
   // the same network as SCL:
   IF "CS1" AND NOT "CS2" AND "BL" THEN "OPERACAO - M3"(); END_IF;
END_REGION

REGION Network 4
   // Verifica nível de pressão do tanque separador
   RUNG wire#powerrail
      "Obtem pressao"(Pressao => #Pressao)
   END_RUNG
   RUNG wire#powerrail
      { S7_Templates := "SrcType := Real" } GE_Contact(in1 := #Pressao, in2 := "L2")
      S_Coil( "LED1" )
   END_RUNG
   RUNG wire#powerrail
      { S7_Templates := "SrcType := Real" } LE_Contact(in1 := #Pressao, in2 := "Lmin")
      R_Coil( "LED1" )
   END_RUNG
   // the same network as SCL:
   "Obtem pressao"(Pressao => #Pressao);
   IF #Pressao >= "L2" THEN "LED1" := TRUE; END_IF;
   IF #Pressao <= "Lmin" THEN "LED1" := FALSE; END_IF;
END_REGION
END_FUNCTION

FUNCTION "OPERACAO - M1" : Void   // FC22, LAD
{ S7_Optimized_Access := 'TRUE' }
VERSION : 0.1
   VAR_TEMP
      "Pressao saida" : Real;   // Pressão na saída do conjunto de compressores
   END_VAR
   VAR_TEMP   // added for the SCL form of the ladder/FBD networks
      _w1 : Bool;
   END_VAR
BEGIN

REGION Network 1
   // Em operação
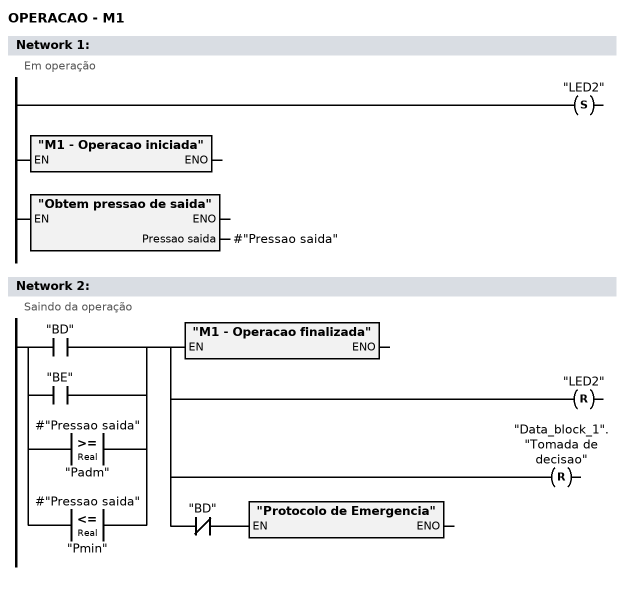
   RUNG wire#powerrail
      S_Coil( "LED2" )
   END_RUNG
   RUNG wire#powerrail
      "M1 - Operacao iniciada"()
   END_RUNG
   RUNG wire#powerrail
      "Obtem pressao de saida"("Pressao saida" => #"Pressao saida")
   END_RUNG
   // the same network as SCL:
   "LED2" := TRUE;
   "M1 - Operacao iniciada"();
   "Obtem pressao de saida"("Pressao saida" => #"Pressao saida");
END_REGION

REGION Network 2
   // Saindo da operação
   RUNG wire#powerrail
      Contact( "BD" )
      wire#w1
      "M1 - Operacao finalizada"()
   END_RUNG
   RUNG wire#powerrail
      Contact( "BE" )
   END_RUNG wire#w1
   RUNG wire#powerrail
      { S7_Templates := "SrcType := Real" } GE_Contact(in1 := #"Pressao saida", in2 := "Padm")
   END_RUNG wire#w1
   RUNG wire#powerrail
      { S7_Templates := "SrcType := Real" } LE_Contact(in1 := #"Pressao saida", in2 := "Pmin")
   END_RUNG wire#w1
   RUNG wire#w1
      R_Coil( "LED2" )
   END_RUNG
   RUNG wire#w1
      R_Coil( "Data_block_1"."Tomada de decisao" )
   END_RUNG
   RUNG wire#w1
      I_Contact( "BD" )
      "Protocolo de Emergencia"()
   END_RUNG
   // the same network as SCL:
   #_w1 := "BD" OR "BE" OR (#"Pressao saida" >= "Padm") OR (#"Pressao saida" <= "Pmin");
   IF #_w1 THEN
       "M1 - Operacao finalizada"();
       "LED2" := FALSE;
       "Data_block_1"."Tomada de decisao" := FALSE;
   END_IF;
   IF #_w1 AND NOT "BD" THEN "Protocolo de Emergencia"(); END_IF;
END_REGION
END_FUNCTION

FUNCTION "OPERACAO - M3" : Void   // FC23, LAD
{ S7_Optimized_Access := 'TRUE' }
VERSION : 0.1
   VAR_TEMP   // added for the SCL form of the ladder/FBD networks
      _w1 : Bool;
   END_VAR
BEGIN

REGION Network 1
   // Em operação
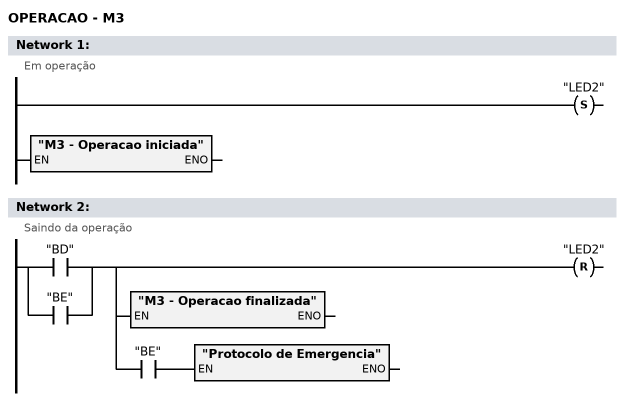
   RUNG wire#powerrail
      S_Coil( "LED2" )
   END_RUNG
   RUNG wire#powerrail
      "M3 - Operacao iniciada"()
   END_RUNG
   // the same network as SCL:
   "LED2" := TRUE;
   "M3 - Operacao iniciada"();
END_REGION

REGION Network 2
   // Saindo da operação
   RUNG wire#powerrail
      Contact( "BD" )
      wire#w1
      R_Coil( "LED2" )
   END_RUNG
   RUNG wire#powerrail
      Contact( "BE" )
   END_RUNG wire#w1
   RUNG wire#w1
      "M3 - Operacao finalizada"()
   END_RUNG
   RUNG wire#w1
      Contact( "BE" )
      "Protocolo de Emergencia"()
   END_RUNG
   // the same network as SCL:
   #_w1 := "BD" OR "BE";
   IF #_w1 THEN
       "LED2" := FALSE;
       "M3 - Operacao finalizada"();
   END_IF;
   IF #_w1 AND "BE" THEN "Protocolo de Emergencia"(); END_IF;
END_REGION
END_FUNCTION

FUNCTION "Atualiza indices" : Void   // FC24, LAD
{ S7_Optimized_Access := 'TRUE' }
VERSION : 0.1
BEGIN

REGION Network 1
   // Movendo sequência 3 1 2
